FUNCTION_BLOCK FB_BeamParamFanout
VAR_INPUT

END_VAR
VAR_OUTPUT
	stBP	:	ST_BeamParams;
END_VAR
VAR
	i_stBP	AT %I* :	ST_BeamParams;
	
	xTxPDO_toggle	AT 	%I* :	BIT;
	xTxPDO_state	AT	%I*	:	BIT;
END_VAR



stBP.xValidToggle;

END_FUNCTION_BLOCK

(* stored: Version 1.1.0.1, ProductVersion 3.1.4024.0
   POU FB_BeamParamFanout: Id {ae70823e-3202-0954-039a-ef27ac7de5b7}, SpecialFunc None *)
